TYPE ST_StationReturn :
STRUCT
	Done	: BOOL;
	stState	: INT;
END_STRUCT
END_TYPE

(* stored: Version 1.1.0.1, ProductVersion 3.1.4024.9
   DUT ST_StationReturn: Id {b3e13514-5f8b-42b7-a8e0-fac6373fac72} *)
